{attribute 'GeneratedUsingTerminal: EL6690-0002-0000'}
{attribute addProperty BoxType "EL6690-0002-0000"}
{attribute addProperty Id "EtcSlaveTerminalBaseStatusAT %I*Status_D30DC33F1InputsEMPTY_STRUCTURE0OutputsEMPTY_STRUCTURE0WcStateAT %I*WcState_9091E0EB2InfoDataAT %I*InfoData_6F19DB2B2"}
{attribute addProperty CRC "2647988852"}
{attribute addProperty Size "5"}
TYPE EL6690_9DD51A74 EXTENDS EtcSlaveTerminalBase :
STRUCT
	{attribute addProperty Name "Status"}
	Status : Status_D30DC33F;
	{attribute addProperty Name "Inputs"}
	Inputs : EMPTY_STRUCTURE;
	{attribute addProperty Name "Outputs"}
	Outputs : EMPTY_STRUCTURE;
	{attribute addProperty Name "WcState"}
	WcState : WcState_9091E0EB;
	{attribute addProperty Name "InfoData"}
	InfoData : InfoData_6F19DB2B;
END_STRUCT
END_TYPE

(* stored: Version 1.2.0.0, ProductVersion 3.1.4024.9
   DUT EL6690_9DD51A74: Id {c82673d7-d1f6-4efd-8842-ae7ba802bbaa} *)
